// TIA Portal project "ARUHAZ_VEZERLES" (V15)

(* hardware
DEVICE "S71500/ET200MP station_1"  S7-1500 station
   slot 0: "Rail_0"  Rack  6ES7 590-1***0-0AA0
   slot 1: "PLC_1"  CPU 1511C-1 PN  6ES7 511-1CK00-0AB0  V2.1
      slot 3: "CPU display_1"  6ES7591-1AA00-0AA0
*)

// ===== PLC "PLC_1"  CPU 1511C-1 PN =====

VAR_GLOBAL   // PLC tag table "Default tag table"
   "System_Byte" AT %MB1 : Byte;
   "FirstScan" AT %M1.0 : Bool;
   "DiagStatusUpdate" AT %M1.1 : Bool;
   "AlwaysTRUE" AT %M1.2 : Bool;
   "AlwaysFALSE" AT %M1.3 : Bool;
   "Clock_Byte" AT %MB0 : Byte;
   "Clock_10Hz" AT %M0.0 : Bool;
   "Clock_5Hz" AT %M0.1 : Bool;
   "Clock_2.5Hz" AT %M0.2 : Bool;
   "Clock_2Hz" AT %M0.3 : Bool;
   "Clock_1.25Hz" AT %M0.4 : Bool;
   "Clock_1Hz" AT %M0.5 : Bool;
   "Clock_0.625Hz" AT %M0.6 : Bool;
   "Clock_0.5Hz" AT %M0.7 : Bool;
END_VAR

VAR_GLOBAL   // PLC tag table "I/O"
   "CONVEYOR_MOVER_BIT_0" AT %I10.0 : Bool;
   "CONVEYOR_MOVER_BIT_1" AT %I10.1 : Bool;
   "CONVEYOR_MOVER_BIT_2" AT %I10.2 : Bool;
   "CONVEYOR_MOVER_BIT_3" AT %I10.3 : Bool;
   "ROBOT_IN_POSTION_BIT_0" AT %I10.4 : Bool;
   "ROBOT_IN_POSTION_BIT_1" AT %I10.5 : Bool;
   "ROBOT_IN_POSTION_BIT_2" AT %I10.6 : Bool;
   "VACUM_IS_OK" AT %I10.7 : Bool;
   "PRODUCT_ID_BIT_0" AT %I11.0 : Bool;
   "PRODUCT_ID_BIT_1" AT %I11.1 : Bool;
   "PRODUCT_ID_BIT_2" AT %I11.2 : Bool;
   "PRODUCT_ID_BIT_3" AT %I11.3 : Bool;
   "INIT_REQUEST" AT %I11.4 : Bool;
   "START_BUTTON" AT %I11.5 : Bool;
   "ORDER_BIT_0" AT %I11.6 : Bool;
   "ORDER_BIT_1" AT %I11.7 : Bool;
   "MOVER_SELECT_BIT_0" AT %Q4.0 : Bool;
   "MOVER_SELECT_BIT_1" AT %Q4.1 : Bool;
   "MOVER_SELECT_BIT_2" AT %Q4.2 : Bool;
   "MOVER_SELECT_BIT_3" AT %Q4.3 : Bool;
   "XTS_CONVEYOR_START" AT %Q4.4 : Bool;
   "ROBOT_POSITION_BIT_SET_0" AT %Q4.5 : Bool;
   "ROBOT_POSITION_BIT_SET_1" AT %Q4.6 : Bool;
   "ROBOT_POSITION_BIT_SET_2" AT %Q4.7 : Bool;
   "ROBOT_MOVEMENT_START" AT %Q5.0 : Bool;
   "VACUM_CONTROL" AT %Q5.1 : Bool;
   "CAMERA_PICTURE_TRIGGER" AT %Q5.2 : Bool;
   "BLUE_INDICATOR_LIGHT" AT %Q5.3 : Bool;
   "YELLOW_INDICATOR_LIGHT" AT %Q5.4 : Bool;
END_VAR

DATA_BLOCK "mainProgram_DB"   // DB1
{ S7_Optimized_Access := 'TRUE' }
VERSION : 0.1
// stored: InstanceOfName mainProgram
"mainProgram"
BEGIN
END_DATA_BLOCK

// folder: System blocks/Program resources

DATA_BLOCK "IEC_Timer_0_DB_2"   // DB2
{ S7_Optimized_Access := 'TRUE' }
AUTHOR : Simatic
FAMILY : IEC
NAME : IEC_TMR
VERSION : 1.0
// stored: InstanceOfName IEC_TIMER
"IEC_TIMER"
BEGIN
END_DATA_BLOCK

DATA_BLOCK "IEC_Timer_0_DB_3"   // DB3
{ S7_Optimized_Access := 'TRUE' }
AUTHOR : Simatic
FAMILY : IEC
NAME : IEC_TMR
VERSION : 1.0
// stored: InstanceOfName IEC_TIMER
"IEC_TIMER"
BEGIN
END_DATA_BLOCK

DATA_BLOCK "IEC_Timer_0_DB_5"   // DB4
{ S7_Optimized_Access := 'TRUE' }
AUTHOR : Simatic
FAMILY : IEC
NAME : IEC_TMR
VERSION : 1.0
// stored: InstanceOfName IEC_TIMER
"IEC_TIMER"
BEGIN
END_DATA_BLOCK

DATA_BLOCK "IEC_Timer_0_DB_4"   // DB5
{ S7_Optimized_Access := 'TRUE' }
AUTHOR : Simatic
FAMILY : IEC
NAME : IEC_TMR
VERSION : 1.0
// stored: InstanceOfName IEC_TIMER
"IEC_TIMER"
BEGIN
END_DATA_BLOCK

DATA_BLOCK "IEC_Timer_0_DB_7"   // DB6
{ S7_Optimized_Access := 'TRUE' }
AUTHOR : Simatic
FAMILY : IEC
NAME : IEC_TMR
VERSION : 1.0
// stored: InstanceOfName IEC_TIMER
"IEC_TIMER"
BEGIN
END_DATA_BLOCK

DATA_BLOCK "IEC_Timer_0_DB_6"   // DB7
{ S7_Optimized_Access := 'TRUE' }
AUTHOR : Simatic
FAMILY : IEC
NAME : IEC_TMR
VERSION : 1.0
// stored: InstanceOfName IEC_TIMER
"IEC_TIMER"
BEGIN
END_DATA_BLOCK

DATA_BLOCK "IEC_Timer_0_DB"   // DB8
{ S7_Optimized_Access := 'TRUE' }
AUTHOR : Simatic
FAMILY : IEC
NAME : IEC_TMR
VERSION : 1.0
// stored: InstanceOfName IEC_TIMER
"IEC_TIMER"
BEGIN
END_DATA_BLOCK

DATA_BLOCK "IEC_Timer_0_DB_8"   // DB9
{ S7_Optimized_Access := 'TRUE' }
AUTHOR : Simatic
FAMILY : IEC
NAME : IEC_TMR
VERSION : 1.0
// stored: InstanceOfName IEC_TIMER
"IEC_TIMER"
BEGIN
END_DATA_BLOCK

DATA_BLOCK "IEC_Timer_0_DB_1"   // DB10
{ S7_Optimized_Access := 'TRUE' }
AUTHOR : Simatic
FAMILY : IEC
NAME : IEC_TMR
VERSION : 1.0
// stored: InstanceOfName IEC_TIMER
"IEC_TIMER"
BEGIN
END_DATA_BLOCK

DATA_BLOCK "IEC_Timer_0_DB_9"   // DB11
{ S7_Optimized_Access := 'TRUE' }
AUTHOR : Simatic
FAMILY : IEC
NAME : IEC_TMR
VERSION : 1.0
// stored: InstanceOfName IEC_TIMER
"IEC_TIMER"
BEGIN
END_DATA_BLOCK

DATA_BLOCK "IEC_Timer_0_DB_10"   // DB12
{ S7_Optimized_Access := 'TRUE' }
AUTHOR : Simatic
FAMILY : IEC
NAME : IEC_TMR
VERSION : 1.0
// stored: InstanceOfName IEC_TIMER
"IEC_TIMER"
BEGIN
END_DATA_BLOCK

DATA_BLOCK "IEC_Timer_0_DB_11"   // DB13
{ S7_Optimized_Access := 'TRUE' }
AUTHOR : Simatic
FAMILY : IEC
NAME : IEC_TMR
VERSION : 1.0
// stored: InstanceOfName IEC_TIMER
"IEC_TIMER"
BEGIN
END_DATA_BLOCK

DATA_BLOCK "IEC_Timer_0_DB_15"   // DB14
{ S7_Optimized_Access := 'TRUE' }
AUTHOR : Simatic
FAMILY : IEC
NAME : IEC_TMR
VERSION : 1.0
// stored: InstanceOfName IEC_TIMER
"IEC_TIMER"
BEGIN
END_DATA_BLOCK

DATA_BLOCK "IEC_Timer_0_DB_12"   // DB17
{ S7_Optimized_Access := 'TRUE' }
AUTHOR : Simatic
FAMILY : IEC
NAME : IEC_TMR
VERSION : 1.0
// stored: InstanceOfName IEC_TIMER
"IEC_TIMER"
BEGIN
END_DATA_BLOCK

DATA_BLOCK "IEC_Timer_0_DB_13"   // DB18
{ S7_Optimized_Access := 'TRUE' }
AUTHOR : Simatic
FAMILY : IEC
NAME : IEC_TMR
VERSION : 1.0
// stored: InstanceOfName IEC_TIMER
"IEC_TIMER"
BEGIN
END_DATA_BLOCK

DATA_BLOCK "IEC_Timer_0_DB_14"   // DB19
{ S7_Optimized_Access := 'TRUE' }
AUTHOR : Simatic
FAMILY : IEC
NAME : IEC_TMR
VERSION : 1.0
// stored: InstanceOfName IEC_TIMER
"IEC_TIMER"
BEGIN
END_DATA_BLOCK

// folder: (top level)

FUNCTION_BLOCK "mainProgram"   // FB1, SCL
{ S7_Optimized_Access := 'TRUE' }
VERSION : 0.1
   VAR_INPUT
      ConveyorMoverBit0 : Bool;
      ConveyorMoverBit1 : Bool;
      ConveyorMoverBit2 : Bool;
      ConveyorMoverBit3 : Bool;
      robotInPostionBit0 : Bool;
      robotInPostionBit1 : Bool;
      robotInPostionBit2 : Bool;
      vacumIsOk : Bool;
      productIdBit0 : Bool;
      productIdBit1 : Bool;
      productIdBit2 : Bool;
      productIdBit3 : Bool;
      initRequest : Bool;
      startButton : Bool;
      orderBit0 : Bool;
      orderBit2 : Bool;
   END_VAR
   VAR_OUTPUT
      moverSelectBit0 : Bool;
      moverSelectBit1 : Bool;
      moverSelectBit2 : Bool;
      moverSelectBit3 : Bool;
      xtsConveyorStart : Bool;
      robotPostionBitSet0 : Bool;
      robotPostionBitSet1 : Bool;
      robotPostionBitSet2 : Bool;
      robotMovementStart : Bool;
      vacumControl : Bool;
      cameraPictureTrigger : Bool;
      blueIndicatorLight : Bool;
      yellowIndicatorLight : Bool;
   END_VAR
   VAR
      moverPostion : Byte;
      "counter" : Int;
      timerRobotOutput : Time;
      timerOutput : Time;
      timerPulse : Bool;
      timerOnDelay : Bool;
      checkRoverBits : Array[0..4] of Bool;
      startRisingEgde : Bool;
      currentState : Int;
      postionMoverArray : Array[0..9] of Byte;
      postionCounter : Int := 0;
      productCode : Array[0..11] of Byte;
      pickCounter : Int := 0;
      productType : Array[0..10] of Int;
      moverPostion_1 : Byte;
      searchForProduct : Int := 1;
      foundProduct : Bool;
      robotBasketPosition : Byte;
      productCounter : Int := 0;
      basketCounter : Int;
      counterCorrection : Int;
   END_VAR
   VAR CONSTANT
      SIGNAL_PULSE : Time := T#250ms;
      SIGNAL_DELAY : Time := T#250ms;
      ROBOT_NONE_POSTION : Byte;
      ROBOT_HOME_POSTION : Byte := 16#1;
      ROBOT_PICK_POSTION : Byte := 16#2;
      ROBOT_BASKET_POSTION_1 : Byte := 16#3;
      ROBOT_BASKET_POSTION_2 : Byte := 16#4;
      ROBOT_BASKET_POSTION_3 : Byte := 16#5;
      ROBOT_BASKET_POSTION_4 : Byte := 16#6;
      ROBOT_INIT_POSTION : Byte := 16#7;
      MOVER_NO_FUNCTION : Byte;
      MOVER_1 : Byte := 16#1;
      MOVER_2 : Byte := 16#2;
      MOVER_3 : Byte := 16#3;
      MOVER_4 : Byte := 16#4;
      MOVER_5 : Byte := 16#5;
      MOVER_6 : Byte := 16#6;
      MOVER_7 : Byte := 16#7;
      MOVER_8 : Byte := 16#8;
      MOVER_9 : Byte := 16#9;
      MOVER_10 : Byte := 16#0A;
      MOVER_INIT : Byte := 16#0F;
      STATE_DEVICE_INIT : Int;
      STATE_DEVICE_SET_CONVEYOR_BITS : Int := 1;
      STATE_DEVICE_START_CONVEYOR : Int := 2;
      STATE_DEVICE_READ_PRODUCT_DATA : Int := 3;
      STATE_DEVICE_START_PICK_AND_PLACE : Int := 4;
      STATE_DEVICE_RESET_TIMERS_CONVEYER : Int := 5;
      STATE_DEVICE_MOVE_PART_TO_PICK_PLACE : Int := 6;
      STATE_DEVICE_START_CONVEYOR_ROBOT_PICK : Int := 7;
      STATE_DEVICE_TRIGGER_CONVEYOR_ROBOT_PICK : Int := 8;
      STATE_DEVICE_TRIGGER_CONVEYOR_ROBOT_PICKUP : Int := 12;
      STATE_DEVICE_SET_ROBOT_PICKUP_POSTION : Int := 9;
      STATE_DEVICE_SEARCH_PRODUCT : Int := 10;
      STATE_DEVICE_MOVE_CONVEYOR_ROBOT_BASKET_1 : Int := 11;
      STATE_DEVICE_TRIGGER_CONVEYOR_ROBOT_BASKET_1 : Int := 13;
      STATE_DEVICE_MOVE_ROBOT_HOME : Int := 14;
      STATE_DEVICE_TRIGGER_ROBOT_HOME : Int := 15;
   END_VAR
   // postionMoverArray[0] := 16#1;
   // postionMoverArray[1] := 16#2;
   // postionMoverArray[2] := 16#3;
   // postionMoverArray[3] := 16#4;
   // postionMoverArray[4] := 16#5;
   // postionMoverArray[5] := 16#6;
   // postionMoverArray[6] := 16#7;
   // postionMoverArray[7] := 16#8;
   // postionMoverArray[8] := 16#9;
   // postionMoverArray[9] := 16#0A;
BEGIN
   CASE #currentState OF
       #STATE_DEVICE_INIT:
           #blueIndicatorLight := TRUE;
           #robotBasketPosition := #ROBOT_BASKET_POSTION_1;

           IF #startButton THEN
               #currentState := #STATE_DEVICE_SET_CONVEYOR_BITS;
           END_IF;

       #STATE_DEVICE_SET_CONVEYOR_BITS:
           "setMoverPostion"(moverPosition := #postionMoverArray[#postionCounter],
                             moverBit0 => #moverSelectBit0,
                             moverBit1 => #moverSelectBit1,
                             moverBit2 => #moverSelectBit2,
                             moverBit3 => #moverSelectBit3);

           "IEC_Timer_0_DB_4".TON(IN := TRUE,
                                  PT := #SIGNAL_DELAY,
                                  Q => #timerOnDelay,
                                  ET => #timerOutput);

           IF #timerOnDelay THEN
               #timerOnDelay := FALSE;
               "IEC_Timer_0_DB_4".TON(IN := FALSE,
                                      PT := #SIGNAL_DELAY);
               #currentState := #STATE_DEVICE_START_CONVEYOR;
           END_IF;

       #STATE_DEVICE_START_CONVEYOR:
           "IEC_Timer_0_DB_6".TP(IN := TRUE,
                                 PT := #SIGNAL_PULSE,
                                 Q => #xtsConveyorStart,
                                 ET => #timerOutput);

           "IEC_Timer_0_DB".TON(IN := TRUE,
                                PT := T#2s,
                                Q => #timerOnDelay,
                                ET => #timerOutput);

           IF #timerOnDelay THEN
               #timerOnDelay := FALSE;
               "IEC_Timer_0_DB".TON(IN := FALSE,
                                    PT := T#3s);
               #currentState := #STATE_DEVICE_READ_PRODUCT_DATA;
           END_IF;

       #STATE_DEVICE_READ_PRODUCT_DATA:
           #cameraPictureTrigger := TRUE;

           "IEC_Timer_0_DB_1".TON(IN := TRUE,
                                  PT := T#350ms,
                                  Q => #timerOnDelay,
                                  ET => #timerOutput);
           IF #timerOnDelay THEN
               #timerOnDelay := FALSE;
               "IEC_Timer_0_DB_1".TON(IN := FALSE,
                                      PT := #SIGNAL_DELAY);

               "getProductTypeAndType"(productBit0 := #productIdBit0,
                                       productBit1 := #productIdBit1,
                                       productBit2 := #productIdBit2,
                                       productBit3 := #productIdBit3,
                                       productCode => #productCode[#postionCounter],
                                       productType => #productType[#postionCounter]);

               #postionCounter := #postionCounter + 1;
               #cameraPictureTrigger := FALSE;

               "IEC_Timer_0_DB_4".TON(IN := FALSE,
                                      PT := #SIGNAL_DELAY);
               "IEC_Timer_0_DB_6".TP(IN := FALSE,
                                     PT := #SIGNAL_PULSE);
               "IEC_Timer_0_DB".TON(IN := FALSE,
                                    PT := T#2s);
               "IEC_Timer_0_DB_1".TON(IN := FALSE,
                                      PT := #SIGNAL_DELAY);

               IF #postionCounter = 10 THEN
                   #xtsConveyorStart := FALSE;
                   "setMoverPostion"(moverPosition := #MOVER_NO_FUNCTION,
                                     moverBit0 => #moverSelectBit0,
                                     moverBit1 => #moverSelectBit1,
                                     moverBit2 => #moverSelectBit2,
                                     moverBit3 => #moverSelectBit3);

                   #currentState := #STATE_DEVICE_SEARCH_PRODUCT;
                   #yellowIndicatorLight := "Clock_0.5Hz";
                   #blueIndicatorLight := FALSE;
                   #postionCounter := 0;
               ELSE
                   #currentState := #STATE_DEVICE_RESET_TIMERS_CONVEYER;
               END_IF;
           END_IF;

       #STATE_DEVICE_RESET_TIMERS_CONVEYER:
           "IEC_Timer_0_DB_4".TON(IN := FALSE,
                                  PT := #SIGNAL_DELAY);
           "IEC_Timer_0_DB_6".TP(IN := FALSE,
                                 PT := #SIGNAL_PULSE);
           "IEC_Timer_0_DB".TON(IN := FALSE,
                                PT := T#3s);
           "IEC_Timer_0_DB_1".TON(IN := FALSE,
                                  PT := #SIGNAL_DELAY);
           #currentState := #STATE_DEVICE_SET_CONVEYOR_BITS;

       #STATE_DEVICE_SEARCH_PRODUCT:
           IF #productCounter = 3 THEN
               #currentState := #STATE_DEVICE_MOVE_ROBOT_HOME;
               RETURN;
           END_IF;

           IF #basketCounter = 0 THEN
               #robotBasketPosition := #ROBOT_BASKET_POSTION_2;
           END_IF;

           IF #basketCounter = 1 THEN
               #robotBasketPosition := #ROBOT_BASKET_POSTION_3;
           END_IF;

           IF #basketCounter = 2 THEN
               #robotBasketPosition := #ROBOT_BASKET_POSTION_4;
               #counterCorrection := 1;
           END_IF;

           IF #basketCounter = 3 THEN
               #currentState := #STATE_DEVICE_INIT;
               RETURN;
           END_IF;

           FOR #counter := 0 TO 9 DO
               IF #productType[#counter] = #searchForProduct THEN
                   #moverPostion := #postionMoverArray[#counter + 1];
                   #productType[#counter] := 0;
                   #currentState := #STATE_DEVICE_MOVE_PART_TO_PICK_PLACE;
                   RETURN;
               ELSE
                   #blueIndicatorLight := TRUE;
               END_IF;
           END_FOR;

       #STATE_DEVICE_MOVE_PART_TO_PICK_PLACE:
           "setMoverPostion"(moverPosition := #moverPostion,
                             moverBit0 => #moverSelectBit0,
                             moverBit1 => #moverSelectBit1,
                             moverBit2 => #moverSelectBit2,
                             moverBit3 => #moverSelectBit3);

           "IEC_Timer_0_DB_12".TON(IN:=TRUE,
                                   PT:=#SIGNAL_DELAY,
                                   Q=>#timerOnDelay,
                                   ET=>#timerOutput);

           IF #timerOnDelay THEN
               "IEC_Timer_0_DB_12".TON(IN := FALSE,
                                       PT := #SIGNAL_DELAY);
               #currentState := #STATE_DEVICE_TRIGGER_CONVEYOR_ROBOT_PICK;
           END_IF;

       #STATE_DEVICE_TRIGGER_CONVEYOR_ROBOT_PICK:
           "IEC_Timer_0_DB_13".TP(IN:=TRUE,
                                  PT:=#SIGNAL_PULSE,
                                  Q=>#xtsConveyorStart,
                                  ET=>#timerOutput);

           "IEC_Timer_0_DB_14".TON(IN:=TRUE,
                                   PT:=T#2s,
                                   Q=>#timerOnDelay,
                                   ET=>#timerOutput);

           IF #timerOnDelay THEN
               "IEC_Timer_0_DB_13".TP(IN := FALSE,
                                      PT := #SIGNAL_PULSE);

               "IEC_Timer_0_DB_14".TON(IN := FALSE,
                                       PT := T#2s);

               #currentState := #STATE_DEVICE_SET_ROBOT_PICKUP_POSTION;
           END_IF;

       #STATE_DEVICE_SET_ROBOT_PICKUP_POSTION:
           "setRobotPostion"(robotPostion := #ROBOT_PICK_POSTION,
                             robotBit0 => #robotPostionBitSet0,
                             robotBit1 => #robotPostionBitSet1,
                             robotBit2 => #robotPostionBitSet2);

           "IEC_Timer_0_DB_2".TON(IN:=TRUE,
                                  PT:=#SIGNAL_DELAY,
                                  Q=>#timerOnDelay,
                                  ET=>#timerOutput);
           IF #timerOnDelay THEN
               "IEC_Timer_0_DB_2".TON(IN:=FALSE,
                                      PT:=#SIGNAL_DELAY);
               #currentState := #STATE_DEVICE_TRIGGER_CONVEYOR_ROBOT_PICKUP;
           END_IF;

       #STATE_DEVICE_TRIGGER_CONVEYOR_ROBOT_PICKUP:
           "IEC_Timer_0_DB_3".TP(IN:=TRUE,
                                 PT:=#SIGNAL_PULSE,
                                 Q=>#robotMovementStart,
                                 ET=>#timerOutput);
           #blueIndicatorLight := TRUE;

           "IEC_Timer_0_DB_5".TON(IN:=TRUE,
                                  PT:=T#2s,
                                  Q=>#timerOnDelay,
                                  ET=>#timerOutput);

           #vacumControl := TRUE;

           IF #timerOnDelay THEN
               "IEC_Timer_0_DB_3".TP(IN := FALSE,
                                     PT := #SIGNAL_PULSE);
               "IEC_Timer_0_DB_5".TON(IN := FALSE,
                                      PT := T#2s);
               #currentState := #STATE_DEVICE_MOVE_CONVEYOR_ROBOT_BASKET_1;
           END_IF;

       #STATE_DEVICE_MOVE_CONVEYOR_ROBOT_BASKET_1:
           "setRobotPostion"(robotPostion := #robotBasketPosition,
                             robotBit0 => #robotPostionBitSet0,
                             robotBit1 => #robotPostionBitSet1,
                             robotBit2 => #robotPostionBitSet2);

           "IEC_Timer_0_DB_7".TON(IN:=TRUE,
                                  PT:=#SIGNAL_DELAY,
                                  Q=>#timerOnDelay,
                                  ET=>#timerOutput);

           IF #timerOnDelay THEN
               "IEC_Timer_0_DB_7".TON(IN := FALSE,
                                      PT := #SIGNAL_DELAY);
               #currentState := #STATE_DEVICE_TRIGGER_CONVEYOR_ROBOT_BASKET_1;
           END_IF;

       #STATE_DEVICE_TRIGGER_CONVEYOR_ROBOT_BASKET_1:
           "IEC_Timer_0_DB_8".TP(IN:=TRUE,
                                 PT:=#SIGNAL_PULSE,
                                 Q=>#robotMovementStart,
                                 ET=>#timerOutput);

           "IEC_Timer_0_DB_9".TON(IN:=TRUE,
                                  PT:=T#2s,
                                  Q=>#timerOnDelay,
                                  ET=>#timerOutput);

           IF #timerOnDelay THEN
               "IEC_Timer_0_DB_8".TP(IN := FALSE,
                                     PT := #SIGNAL_PULSE);

               "IEC_Timer_0_DB_9".TON(IN := FALSE,
                                      PT := T#2s);

               #productCounter := #productCounter + 1;
               #vacumControl := FALSE;
               #currentState := #STATE_DEVICE_SEARCH_PRODUCT;
               #searchForProduct := #searchForProduct + 1;
           END_IF;

       #STATE_DEVICE_MOVE_ROBOT_HOME:
           "setRobotPostion"(robotPostion := #ROBOT_HOME_POSTION,
                             robotBit0 => #robotPostionBitSet0,
                             robotBit1 => #robotPostionBitSet1,
                             robotBit2 => #robotPostionBitSet2);

           "IEC_Timer_0_DB_10".TON(IN:=TRUE,
                                   PT:=#SIGNAL_DELAY,
                                   Q=>#timerOnDelay,
                                   ET=>#timerOutput);

           IF #timerOnDelay THEN
               "IEC_Timer_0_DB_10".TON(IN := FALSE,
                                       PT := #SIGNAL_DELAY);
               #currentState := #STATE_DEVICE_TRIGGER_ROBOT_HOME;
           END_IF;

       #STATE_DEVICE_TRIGGER_ROBOT_HOME:
           "IEC_Timer_0_DB_11".TP(IN:=TRUE,
                                  PT:=#SIGNAL_PULSE,
                                  Q=>#robotMovementStart,
                                  ET=>#timerOutput);

           "IEC_Timer_0_DB_15".TON(IN:=TRUE,
                                   PT:=T#1s,
                                   Q=>#timerOnDelay,
                                   ET=>#timerOutput);

           IF #timerOnDelay THEN
               "IEC_Timer_0_DB_11".TP(IN := FALSE,
                                      PT := #SIGNAL_PULSE);

               "IEC_Timer_0_DB_15".TON(IN := FALSE,
                                       PT := T#1s);

               #currentState := #STATE_DEVICE_SEARCH_PRODUCT;
               #basketCounter := #basketCounter + 1;
               #productCounter := 0;
               #searchForProduct := 1;
           END_IF;
   END_CASE;
END_FUNCTION_BLOCK

FUNCTION "setRobotPostion" : Void   // FC1, SCL
{ S7_Optimized_Access := 'TRUE' }
VERSION : 0.1
   VAR_INPUT
      robotPostion : Byte;
   END_VAR
   VAR_OUTPUT
      robotBit0 : Bool;
      robotBit1 : Bool;
      robotBit2 : Bool;
   END_VAR
BEGIN
   #robotBit0 := (#robotPostion AND BYTE#16#01) <> BYTE#0;
   #robotBit1 := (#robotPostion AND BYTE#16#02) <> BYTE#0;
   #robotBit2 := (#robotPostion AND BYTE#16#04) <> BYTE#0;
END_FUNCTION

FUNCTION "getProductTypeAndType" : Void   // FC2, SCL
{ S7_Optimized_Access := 'TRUE' }
VERSION : 0.1
   VAR_INPUT
      productBit0 : Bool;
      productBit1 : Bool;
      productBit2 : Bool;
      productBit3 : Bool;
   END_VAR
   VAR_OUTPUT
      productCode : Byte;
      productType : Int;
   END_VAR
   VAR_TEMP
      tempCode : Byte;
   END_VAR
   VAR CONSTANT
      NO_FUNCTION : Byte;
      PRODUCT_1 : Byte := 16#1;
      PRODUCT_2 : Byte := 16#2;
      PRODUCT_3 : Byte := 16#3;
      PRODUCT_4 : Byte := 16#4;
      PRODUCT_5 : Byte := 16#5;
      PRODUCT_6 : Byte := 16#6;
      PRODUCT_7 : Byte := 16#7;
      PRODUCT_8 : Byte := 16#8;
      PRODUCT_9 : Byte := 16#9;
      PRODUCT_10 : Byte := 16#0A;
      NO_READ : Byte := 16#0F;
      TYPE_NONE : Int;
      TYPE_ELECTRONIC : Int := 1;
      TYPE_PNEUMATIC : Int := 2;
      TYPE_MECHANICAL : Int := 3;
   END_VAR
BEGIN
   #tempCode := BYTE#16#00;
   IF #productBit0 THEN
       #tempCode := #tempCode OR BYTE#16#01;
   END_IF;

   IF #productBit1 THEN
       #tempCode := #tempCode OR BYTE#16#02;
   END_IF;

   IF
       #productBit2 THEN #tempCode := #tempCode OR BYTE#16#04;
   END_IF;
   IF
       #productBit3 THEN #tempCode := #tempCode OR BYTE#16#08;
   END_IF;

   #productCode := #tempCode;

   // case numbers are products from 1 - 10
   CASE BYTE_TO_INT(#tempCode) OF
       1:  #productType := #TYPE_ELECTRONIC;
       2:  #productType := #TYPE_PNEUMATIC;
       3:  #productType := #TYPE_MECHANICAL;
       4:  #productType := #TYPE_ELECTRONIC;
       5:  #productType := #TYPE_PNEUMATIC;
       6:  #productType := #TYPE_MECHANICAL;
       7:  #productType := #TYPE_ELECTRONIC;
       8:  #productType := #TYPE_PNEUMATIC;
       9:  #productType := #TYPE_MECHANICAL;
       10: #productType := #TYPE_PNEUMATIC;
       ELSE: #productType := #TYPE_NONE;
   END_CASE;
END_FUNCTION

FUNCTION "setMoverPostion" : Void   // FC3, SCL
{ S7_Optimized_Access := 'TRUE' }
VERSION : 0.1
   VAR_INPUT
      moverPosition : Byte;
   END_VAR
   VAR_OUTPUT
      moverBit0 : Bool;
      moverBit1 : Bool;
      moverBit2 : Bool;
      moverBit3 : Bool;
   END_VAR
BEGIN
   #moverBit0 := (#moverPosition AND BYTE#16#01) <> BYTE#0;
   #moverBit1 := (#moverPosition AND BYTE#16#02) <> BYTE#0;
   #moverBit2 := (#moverPosition AND BYTE#16#04) <> BYTE#0;
   #moverBit3 := (#moverPosition AND BYTE#16#08) <> BYTE#0;
END_FUNCTION

ORGANIZATION_BLOCK "Main"   // OB1, LAD, ProgramCycle
TITLE = "Main Program Sweep (Cycle)"
{ S7_Optimized_Access := 'TRUE' }
VERSION : 0.1
   VAR_INPUT
      Initial_Call : Bool;   // Initial call of this OB
      Remanence : Bool;   // =True, if remanent data are available
   END_VAR
BEGIN

REGION Network 1
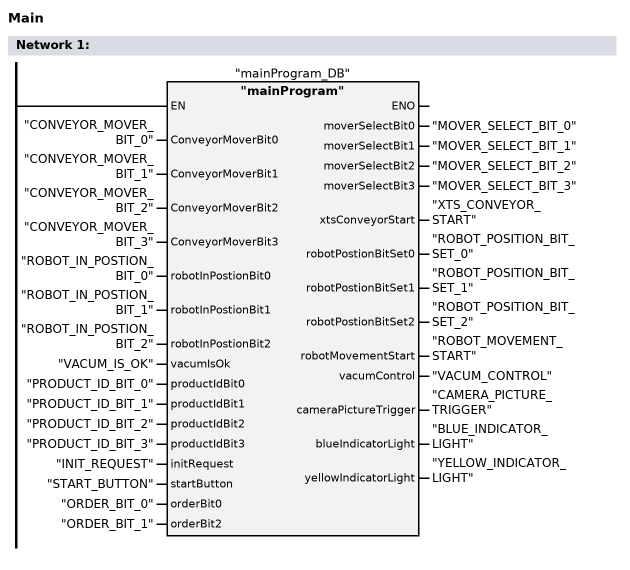
   RUNG wire#powerrail
      "mainProgram_DB"(ConveyorMoverBit0 := "CONVEYOR_MOVER_BIT_0", ConveyorMoverBit1 := "CONVEYOR_MOVER_BIT_1", ConveyorMoverBit2 := "CONVEYOR_MOVER_BIT_2", ConveyorMoverBit3 := "CONVEYOR_MOVER_BIT_3", robotInPostionBit0 := "ROBOT_IN_POSTION_BIT_0", robotInPostionBit1 := "ROBOT_IN_POSTION_BIT_1", robotInPostionBit2 := "ROBOT_IN_POSTION_BIT_2", vacumIsOk := "VACUM_IS_OK", productIdBit0 := "PRODUCT_ID_BIT_0", productIdBit1 := "PRODUCT_ID_BIT_1", productIdBit2 := "PRODUCT_ID_BIT_2", productIdBit3 := "PRODUCT_ID_BIT_3", initRequest := "INIT_REQUEST", startButton := "START_BUTTON", orderBit0 := "ORDER_BIT_0", orderBit2 := "ORDER_BIT_1", moverSelectBit0 => "MOVER_SELECT_BIT_0", moverSelectBit1 => "MOVER_SELECT_BIT_1", moverSelectBit2 => "MOVER_SELECT_BIT_2", moverSelectBit3 => "MOVER_SELECT_BIT_3", xtsConveyorStart => "XTS_CONVEYOR_START", robotPostionBitSet0 => "ROBOT_POSITION_BIT_SET_0", robotPostionBitSet1 => "ROBOT_POSITION_BIT_SET_1", robotPostionBitSet2 => "ROBOT_POSITION_BIT_SET_2", robotMovementStart => "ROBOT_MOVEMENT_START", vacumControl => "VACUM_CONTROL", cameraPictureTrigger => "CAMERA_PICTURE_TRIGGER", blueIndicatorLight => "BLUE_INDICATOR_LIGHT", yellowIndicatorLight => "YELLOW_INDICATOR_LIGHT")
   END_RUNG
   // the same network as SCL:
   "mainProgram_DB"(ConveyorMoverBit0 := "CONVEYOR_MOVER_BIT_0",   // "mainProgram"
                    ConveyorMoverBit1 := "CONVEYOR_MOVER_BIT_1",
                    ConveyorMoverBit2 := "CONVEYOR_MOVER_BIT_2",
                    ConveyorMoverBit3 := "CONVEYOR_MOVER_BIT_3",
                    robotInPostionBit0 := "ROBOT_IN_POSTION_BIT_0",
                    robotInPostionBit1 := "ROBOT_IN_POSTION_BIT_1",
                    robotInPostionBit2 := "ROBOT_IN_POSTION_BIT_2",
                    vacumIsOk := "VACUM_IS_OK",
                    productIdBit0 := "PRODUCT_ID_BIT_0",
                    productIdBit1 := "PRODUCT_ID_BIT_1",
                    productIdBit2 := "PRODUCT_ID_BIT_2",
                    productIdBit3 := "PRODUCT_ID_BIT_3",
                    initRequest := "INIT_REQUEST",
                    startButton := "START_BUTTON",
                    orderBit0 := "ORDER_BIT_0",
                    orderBit2 := "ORDER_BIT_1",
                    moverSelectBit0 => "MOVER_SELECT_BIT_0",
                    moverSelectBit1 => "MOVER_SELECT_BIT_1",
                    moverSelectBit2 => "MOVER_SELECT_BIT_2",
                    moverSelectBit3 => "MOVER_SELECT_BIT_3",
                    xtsConveyorStart => "XTS_CONVEYOR_START",
                    robotPostionBitSet0 => "ROBOT_POSITION_BIT_SET_0",
                    robotPostionBitSet1 => "ROBOT_POSITION_BIT_SET_1",
                    robotPostionBitSet2 => "ROBOT_POSITION_BIT_SET_2",
                    robotMovementStart => "ROBOT_MOVEMENT_START",
                    vacumControl => "VACUM_CONTROL",
                    cameraPictureTrigger => "CAMERA_PICTURE_TRIGGER",
                    blueIndicatorLight => "BLUE_INDICATOR_LIGHT",
                    yellowIndicatorLight => "YELLOW_INDICATOR_LIGHT");
END_REGION
END_ORGANIZATION_BLOCK